TYPE DUT_CMD_ForceCompletedBatch:
STRUCT  
	return_value	: DINT;
	Id	: STRING(50);
END_STRUCT
END_TYPE

(* stored: Version 1.1.0.1, ProductVersion 3.1.4024.15
   DUT DUT_CMD_ForceCompletedBatch: Id {3391f245-3049-4a5f-b564-159ae10966e1} *)
